TYPE "HU_Pump_Config"
VERSION : 0.1
// Block: HU_Pump_Config
   STRUCT
      SafetyCutOffValveExist : Bool;
      StandbyValveExist : Bool;
      OilPumpContactotFeedbackTimeOut : Time;
   END_STRUCT;

END_TYPE
